Universal Robots PolyScope program: T00 Basic.urp

Program T00 Basic (installation=default directory=/programs createdIn=5.9.1.1031110 lastSavedIn=5.9.1.1031110 robotSerialNumber=20195501059)
Calibrated DH parameters: a=[0.000146, -0.418764, -0.053981, 0.000058, -0.000023, 0]; d=[0.162545, 37.319448, -206.067439, 168.881546, 0.09955, 0.099464]; alpha=[1.57004, -0.001979, 0.002304, 1.570607, -1.57066, 0]; deltaTheta=[0, -0.174616, -1.258233, 1.432844, -0.000001, 0]
BeforeStart
  start_p := get_actual_tcp_pose()
  MoveJ speed 60 deg/s, acceleration 80 deg/s^2 (useActiveTCP=true) feature=Base
    Waypoint Waypoint (Variable): variable=start_p
Robot Program (runOnlyOnce=true)
  MoveJ speed 60 deg/s, acceleration 80 deg/s^2 (useActiveTCP=true) feature=Base
    Waypoint Waypoint_1: TCP in base x=153.849 y=-567.885 z=95.237 mm, rx=2.2517 ry=2.1906 rz=0.0001 rad; joints [92.011, -71.611, 101.775, -120.157, 270.027, 93.606] deg; TCP offset x=0 y=0 z=174 mm, rx=0 ry=0 rz=0 rad
  URCap Olis Teleop (Olis Teleop, Olis Robotics)
  current_p := get_actual_tcp_pose()
  MoveJ speed 60 deg/s, acceleration 80 deg/s^2 (useActiveTCP=true) feature=Base
    Waypoint Waypoint (Variable): variable=current_p
  SuppressedNode
    Wait Sleep waitTime=1
  MoveL speed 250 mm/s, acceleration 1200 mm/s^2 (useActiveTCP=true) feature=Base
    Waypoint Waypoint_2: TCP in base x=135.121 y=-561.417 z=95.227 mm, rx=2.2518 ry=2.1906 rz=0.0001 rad; joints [90.133, -72.944, 103.616, -120.662, 270.031, 91.73] deg
    Waypoint Waypoint_1: TCP in base x=153.849 y=-567.885 z=95.237 mm, rx=2.2517 ry=2.1906 rz=0.0001 rad; joints [92.011, -71.611, 101.775, -120.157, 270.027, 93.606] deg
